// TIA Portal V20 export
// export: Created 2025-09-12T17:59:00.0000000Z, ExportSetting WithDefaults
FUNCTION_BLOCK "FB300_EM_Heating"   // FB, SCL
TITLE = EM-300: Heating Control
AUTHOR : Dallas Levine
VERSION : 0.1
// This block contains all logic for the Heating Equipment Module (EM-300).
// stored: AutoNumber true, IsRetain false
   VAR_INPUT
      Enable : Bool;   // Enables the block's execution.
   END_VAR
   VAR
      UDT : "UDT300_EM_Heating";   // The data interface for the Heating Equipment Module.
   END_VAR
BEGIN
   REGION Placeholder for SCL Code 

   END_REGION
END_FUNCTION_BLOCK
